// TIA Portal V19 export
TYPE "ItemTimer_UDT"
   STRUCT
      SpareByte : Byte;
      fb_timer : Byte;
   END_STRUCT;
END_TYPE
